Universal Robots PolyScope program: cottonHeatOn.urp

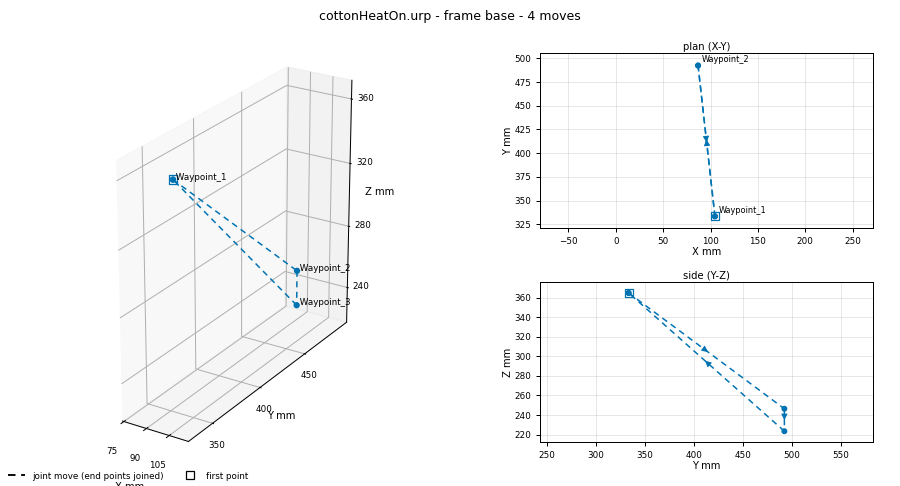
[picture p0: tool path of cottonHeatOn.urp in frame base, 4 of 6 moves have a stored position in this frame; points joined in program order, loops and branches not executed]
Program cottonHeatOn (installation=default directory=/programs/DavidMelin createdIn=5.12.4.1101661 lastSavedIn=5.12.4.1101661 robotSerialNumber=20225502378)
Calibrated DH parameters: a=[0.00022, -0.425328, -0.389701, 0.000059, 0.000065, 0]; d=[0.162608, 0.803456, 9.992211, -10.662202, 0.099702, 0.099559]; alpha=[1.570756, 0.001543, 0.004316, 1.570651, -1.570122, 0]; deltaTheta=[0, 0.002917, 0.116094, -0.119008, 0, -0.000001]
Robot Program (runOnlyOnce=true)
  MoveJ speed 60 deg/s, acceleration 80 deg/s^2 (useActiveTCP=true) feature=Base
    Waypoint Waypoint (Variable): variable=cotonHomePos
  URCap Gripper (Robotiq_Grippers, Robotiq Inc.) dataModel(position=100.0, force=0.0, speed=0.0, positionInDouble=100.0, forceInDouble=0.0, speedInDouble=0.0, slaveIds=[9], blocking=true)
  MoveJ speed 60 deg/s, acceleration 80 deg/s^2 (useActiveTCP=true) feature=Base
    Waypoint Waypoint_1: TCP in base x=104.657 y=333.28 z=364.781 mm, rx=-2.4906 ry=0.0958 rz=-0.1131 rad; joints [98.535, -64.729, -139.702, -29.679, 79.086, 9.451] deg
    Waypoint Waypoint_2: TCP in base x=86.856 y=492.404 z=246.455 mm, rx=-2.3949 ry=0.1183 rz=-0.0956 rad; joints [97.805, -104.935, -129.813, 6.213, 78.977, 9.441] deg
    Waypoint Waypoint_3: TCP in base x=86.848 y=492.416 z=223.524 mm, rx=-2.3949 ry=0.1183 rz=-0.0956 rad; joints [97.805, -108.318, -130.629, 10.412, 78.962, 9.444] deg
    Waypoint Waypoint_4: TCP in base x=104.669 y=333.277 z=364.778 mm, rx=-2.4906 ry=0.0958 rz=-0.1132 rad; joints [98.533, -64.729, -139.703, -29.679, 79.085, 9.451] deg
    Waypoint Waypoint (Variable): variable=cotonHomePos
